# EPICS StreamDevice protocol: protocols/moxa.proto
# For getting the US and DS measurements fro theKeyenceLS7501 throug a Moxa unit

ExtraInput = Ignore;
ReadTimeout = 500;
OutTerminator = "";
InTerminator = "";
Separator = "";

getUS
{
  out "M1,0" CR;
  in  "M1,%f" CR;
}

getDS
{
  out "M2,0" CR;
  in  "M2,%f" CR;
}
